PROGRAM MAIN
VAR
	mErrACK AT %Q*	: BOOL;
	mRun AT %Q*		: BOOL;
	
END_VAR

mRun := True;

END_PROGRAM

(* stored: Version 1.1.0.1, ProductVersion 3.1.4022.18
   POU MAIN: Id {8a9b52c3-21a9-4800-996e-a0c3716d80ae}, SpecialFunc None *)
